FUNCTION F_HaveDifferentIDs : BOOL
VAR_INPUT
    msg1: ST_MsgToPLC;
    msg2: ST_MsgToPLC;
END_VAR

(* First compare the fields most likely to have changed. *)
F_HaveDifferentIDs :=
    (msg1.dtime 	<> msg2.dtime) OR_ELSE
    (msg1.sequence 	<> msg2.sequence) OR_ELSE
    (msg1.lowUUID 	<> msg2.lowUUID) OR_ELSE
    (msg1.highUUID	<> msg2.highUUID);

END_FUNCTION

(* stored: Version 1.1.0.1, ProductVersion 3.1.4022.18
   POU F_HaveDifferentIDs: Id {efee81a6-e141-448b-8c77-517e06ad4102}, SpecialFunc None *)
